VAR_GLOBAL CONSTANT
	iSLAVEADDR_ARR_SIZE	: UDINT := 256;
    ESC_MAX_PORTS : UINT := 3; // Maximum number of ports (4) on ESC
END_VAR

(* stored: Version 1.1.0.1, ProductVersion 3.1.4022.18
   GVL Global_Variables_EtherCAT: Id {d76f2eaf-f0c3-42c2-8317-22c7ba689cf7} *)
